PROGRAM ArmPickTransferCtrl_General
VAR
	fbGenerateArmPickTransferBit_Arm1Horz		: fbV2_GenerateArmPickTransferBit;

END_VAR

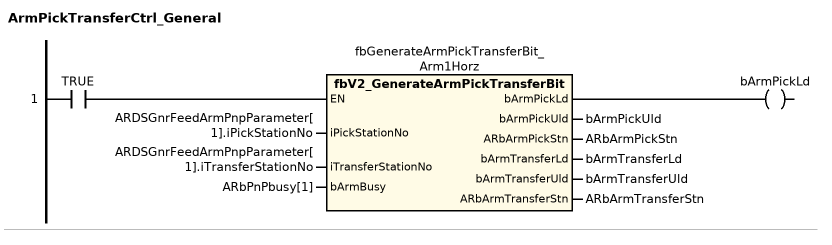
// NETWORK 1
fbGenerateArmPickTransferBit_Arm1Horz(
    iPickStationNo := ARDSGnrFeedArmPnpParameter[1].iPickStationNo,
    iTransferStationNo := ARDSGnrFeedArmPnpParameter[1].iTransferStationNo,
    bArmBusy := ARbPnPbusy[1],
    bArmPickUld => bArmPickUld,
    ARbArmPickStn => ARbArmPickStn,
    bArmTransferLd => bArmTransferLd,
    bArmTransferUld => bArmTransferUld,
    ARbArmTransferStn => ARbArmTransferStn); // fbV2_GenerateArmPickTransferBit
bArmPickLd := fbGenerateArmPickTransferBit_Arm1Horz.bArmPickLd;

END_PROGRAM

(* stored: Version 1.1.0.1, ProductVersion 3.1.4024.12
   POU ArmPickTransferCtrl_General: Id {fad943e3-e0db-4cae-b7f2-127f51fb5b9a}, SpecialFunc None *)
